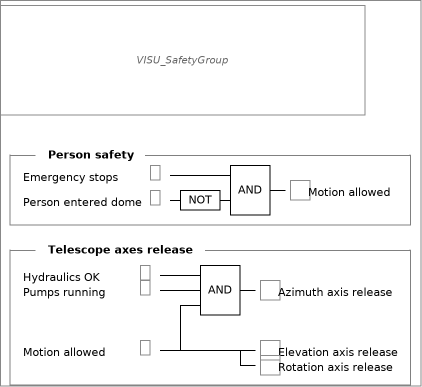
VISUALIZATION VISU_SafetyMotionBlocking  // 422x387
VAR_IN_OUT
	ref : SafetyMotionBlocking;
    ref_hydraulics : SafetyHydraulics;
    ref_emergencyStops : SafetyEmergencyStops;
    ref_domeAccess : SafetyDomeAccess;
    widget : SafetyMotionBlockingWidget;
END_VAR
    Polyline (145,155) (410,155) (410,225) (10,225) (10,155) (35,155)
    Polyline (205,250) (410,250) (410,385) (10,385) (10,250) (35,250)
    Frame (260,280 20x20)
        shows VISU_State_red_green(state := ref.telescopeAzimuthReleaseOK)
    Frame (140,265 10x15)
        shows VISU_State_red_green(state := ref_hydraulics.allOK)
    Label (20,270 100x15), "Hydraulics OK"
    Label (20,285 120x15), "Pumps running"
    Rectangle (200,265 40x50), "AND"
    Line (160,275) (200,275), colour toggle: ref_hydraulics.allOK
    Label (275,280 145x25), "Azimuth axis release"
    Label (45,240 150x20), "Telescope axes release"
    Line (240,290) (255,290), colour toggle: ref.telescopeAzimuthReleaseOK
    Frame (140,280 10x15)
        shows VISU_State_gray_green(state := ref_hydraulics.pumpsRunning)
    Line (160,290) (200,290), colour toggle: ref_hydraulics.pumpsRunning
    Frame (140,340 10x15)
        shows VISU_State_red_green(state := ref.motionAllowed)
    Line (160,350) (255,350), colour toggle: ref.motionAllowed
    Label (20,345 120x15), "Motion allowed"
    Frame (0,5 365x110)
        shows VISU_SafetyGroup(statusWidget := widget.actualStatus, comError := ref.groupComError, fbError := ref.groupFbError, outError := ref.groupOutError, reset := ref.processes.reset)
    Frame (290,180 20x20)
        shows VISU_State_red_green(state := ref.motionAllowed)
    Rectangle (230,165 40x50), "AND"
    Label (305,180 100x25), "Motion allowed"
    Label (45,145 150x20), "Person safety"
    Line (270,190) (285,190), colour toggle: ref.motionAllowed
    Frame (150,165 10x15)
        shows VISU_State_red_green(state := ref_emergencyStops.allOK)
    Line (170,175) (230,175), colour toggle: ref_emergencyStops.allOK
    Label (20,170 120x15), "Emergency stops"
    Label (20,195 130x15), "Person entered dome"
    Rectangle (180,190 40x20), "NOT"
    Line (220,200) (230,200), colour toggle: ref_domeAccess.personHasEntered
    Frame (150,190 10x15)
        shows VISU_State_gray_red(state := ref_domeAccess.personHasEntered)
    Line (170,200) (180,200), colour toggle: ref_domeAccess.personHasEntered
    Line (180,305) (180,350), colour toggle: ref.motionAllowed
    Line (180,305) (200,305), colour toggle: ref.motionAllowed
    Frame (260,340 20x20)
        shows VISU_State_red_green(state := ref.telescopeElevationReleaseOK)
    Label (275,340 145x25), "Elevation axis release"
    Frame (260,355 20x20)
        shows VISU_State_red_green(state := ref.telescopeRotationReleaseOK)
    Label (275,355 145x25), "Rotation axis release"
    Line (240,350) (240,365), colour toggle: ref.motionAllowed
    Line (240,365) (255,365), colour toggle: ref.motionAllowed
END_VISUALIZATION

(* stored: Version 1.1.0.1, ProductVersion 3.1.4019.2
   Visu VISU_SafetyMotionBlocking: Id {a0494e0f-1e4f-42b2-87bb-12fb1ac25a0b} *)
